// TIA Portal V19 export
TYPE "lexchangetray_typeUnEmn_toRollerReq"
// Type: Bool
// stored: Access Published
   STRUCT
      outFeedReq : Bool;   // 请求排料
   END_STRUCT;
END_TYPE
